RoboDK station: Concept_2.rdk

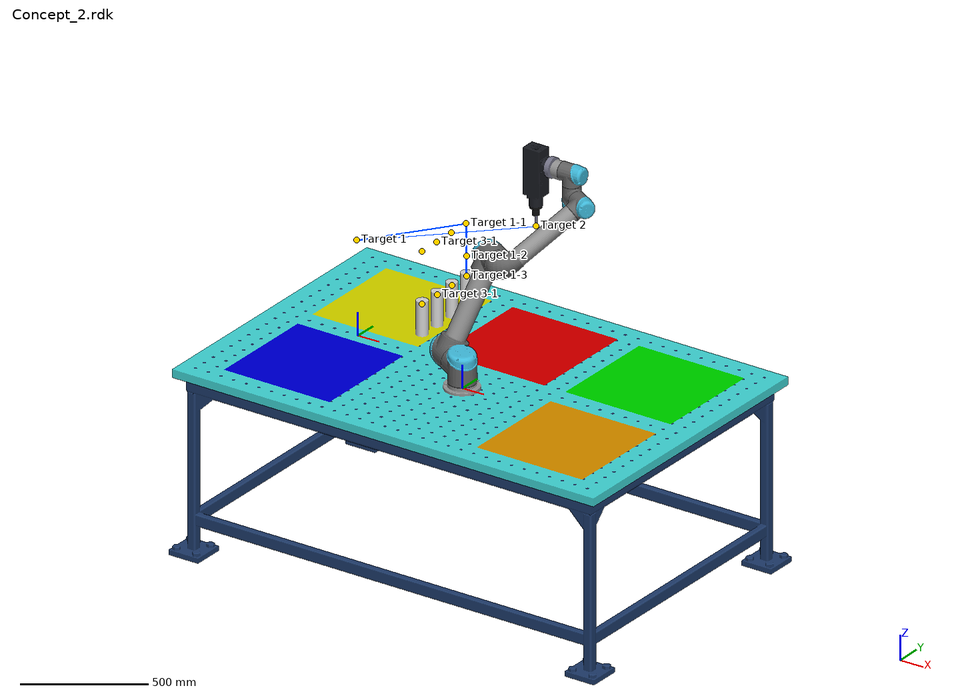
[picture v0: the station drawn from its stored meshes, robots at their saved joint values, targets as dots, program paths as lines]
Station Concept_2 (saved by RoboDK 5.3.4). Poses are relative to the parent item; angles as X-Y-Z fixed-axis rotations.
  - frame UR5 Base at (0, 0, 0) mm
    - robot UR5: 6 axes, payload 5 kg, reach 850 mm, repeatability 0.1 mm, weight 18.4 kg
        modified DH rows (alpha deg, a mm, theta deg, d mm): 0, 0, 0, 89.2; 90, 0, 180, 0; 0, 425, 0, 0; 0, 392.43, 0, 109; -90, 0, 0, 93.65; 90, 0, 180, 82
        joint limits [-360, -360, -360, -360, -360, -360] to [360, 360, 360, 360, 360, 360]; home [0, -90, -90, 0, 90, 0]; saved at [238.928, -64.181, 31.334, 213.045, 31.083, -270.699]
      - tool Spindle, TCP at (278.6, 0, 90) mm, rotated rx 0 ry 90 rz 0 deg, size 85 x 346.5 x 128 mm
  - frame Work Space at (-600, 150, 0) mm
    - object Cell Frame 3.5m at (0, 0, 0) mm, size 2018.1 x 1282.7 x 844.7 mm, geometry from Cell-Frame-3.5m.sld
    - object Table 2000x1200x800 at (0, 0, 0) mm, size 2020 x 1340 x 800 mm, geometry from Table-2000mmx1200mmx800mm.sld
  - frame Tubes at (0, 0, 0) mm
    - object Cylinder 1 at (0, 0, 0) mm, size 50 x 50 x 150 mm, geometry from Cylinder-100mmx300mm.sld
    - target Target 1-1 (Cartesian target) at (-400, 600, 360.05) mm, rotated rx -179.47 ry 0.1 rz 0.01 deg; joints [120.663, -126.918, -35.935, 343.053, 149.348, -270.358] of UR5
    - target Target 1-2 (Cartesian target) at (-400.25, 601.32, 217.71) mm, rotated rx -179.47 ry 0.1 rz 0.01 deg; joints [281.029, -55.383, 60.736, 174.112, -11.019, -270.006] of UR5
    - target Target 1-3 (Cartesian target) at (-400.41, 602.11, 131.43) mm, rotated rx -179.47 ry 0.1 rz 0.01 deg; joints [281.029, -52.827, 69.376, 162.917, -11.019, -270.006] of UR5
    - object Cylinder 2 at (0, 0, 0) mm, size 50 x 50 x 150 mm, geometry from Cylinder-100mmx300mm.sld
    - target Target 2-1 (Cartesian target) at (-400, 500, 360.05) mm, rotated rx -179.47 ry 0.1 rz 0.01 deg; joints [126.07, -110.39, -61.242, 351.805, 143.94, -270.39] of UR5
    - target Target 2-2 (Cartesian target) at (-400.41, 502.11, 131.43) mm, rotated rx -179.47 ry 0.1 rz 0.01 deg; joints [283.074, -64.973, 88.751, 155.77, -13.063, -270.09] of UR5
    - object Cylinder 3 at (0, 0, 0) mm, size 50 x 50 x 150 mm, geometry from Cylinder-100mmx300mm.sld
    - target Target 3-1 (Cartesian target) at (-400, 400, 360.05) mm, rotated rx -179.47 ry 0.1 rz 0.01 deg; joints [133.556, -97.311, -77.728, 355.187, 136.455, -270.423] of UR5
    - target Target 3-1 (Cartesian target) at (-400.41, 402.11, 131.43) mm, rotated rx -179.47 ry 0.1 rz 0.01 deg; joints [285.993, -76.138, 104.39, 151.377, -15.983, -270.173] of UR5
    - object Cylinder 4 at (0, 0, 0) mm, size 50 x 50 x 150 mm, geometry from Cylinder-100mmx300mm.sld
    - target Target 4-1 (Cartesian target) at (-400, 300, 360.05) mm, rotated rx -179.47 ry 0.1 rz 0.01 deg; joints [144.332, -85.591, -89.769, 355.486, 125.679, -270.457] of UR5
    - target Target 4-2 (Cartesian target) at (-400.41, 302.12, 131.43) mm, rotated rx -179.47 ry 0.1 rz 0.01 deg; joints [290.431, -87.073, 117.304, 149.477, -20.421, -270.256] of UR5
  - frame Zones at (0, 0, 0) mm
    - object Raw Material at (0, 0, 0) mm, size 500 x 500 x 0 mm, geometry from Square.sld
      - object Raw Material at (0, 0, 0) mm, size 500 x 500 x 0 mm, geometry from Square.sld
    - object Solution at (0, 0, 0) mm, size 500 x 500 x 0 mm, geometry from Square.sld
    - object Processing at (0, 0, 0) mm, size 500 x 500 x 0 mm, geometry from Square.sld
    - object Cleaning at (0, 0, 0) mm, size 500 x 500 x 0 mm, geometry from Square.sld
    - object Storage at (0, 0, 0) mm, size 500 x 500 x 0 mm, geometry from Square.sld
    - target Target 1 (Cartesian target) at (-500, 0.36, 500) mm, rotated rx -179.47 ry 0.1 rz 0.01 deg; joints [340.942, -95.86, 69.759, 205.993, -70.931, -270.495] of UR5
    - target Target 2 (Cartesian target) at (0, 500, 500) mm, rotated rx -179.47 ry 0.1 rz 0.01 deg; joints [238.928, -64.181, 31.334, 213.045, 31.083, -270.699] of UR5
  - program 程序1 (9 instructions, listed below)
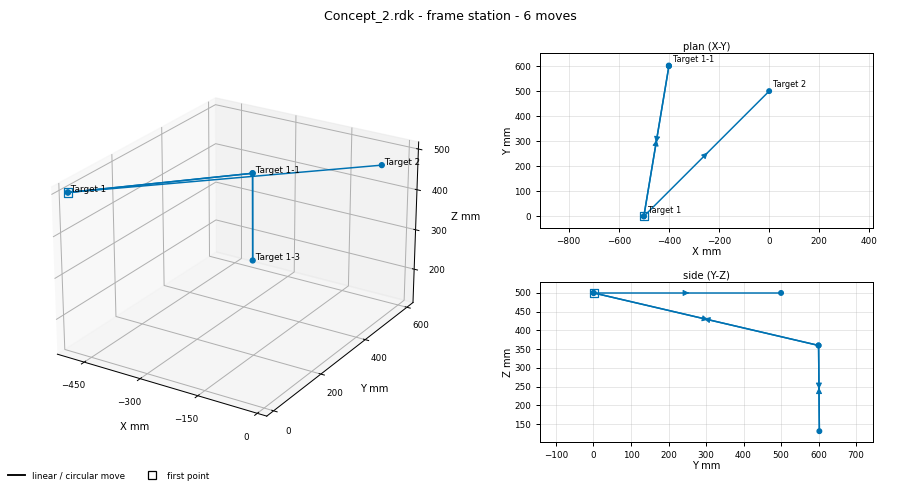
[picture p0: tool path of Concept_2.rdk in frame station, 6 of 6 moves have a stored position in this frame; points joined in program order, loops and branches not executed]

--- program 程序1 (robot UR5) ---
  替换物体
  设置参考: Zones
  设置工具: Spindle
  MoveJ (Target 1)
  MoveL (Target 1-1)
  MoveL (Target 1-3)
  MoveL (Target 1-1)
  MoveL (Target 1)
  MoveL (Target 2)
